FUNCTION_BLOCK EL2596
VAR
	{attribute addProperty Name "WcState"}
	_wcState : WcStateInputToggle;
	{attribute addProperty Name "Info data"}
	_infoData : InfoDataAds;
	_io : EL2596_Data;
END_VAR

PROPERTY IO : REFERENCE TO EL2596_Data
GET
IO REF= _io;
END_GET
END_PROPERTY

PROPERTY WcState : REFERENCE TO WcStateInputToggle
GET
WcState REF= _wcState;
END_GET
END_PROPERTY

END_FUNCTION_BLOCK

(* stored: Version 1.1.0.1, ProductVersion 3.1.4024.9
   POU EL2596: Id {c7ce0382-a06f-0c21-033a-7edddd5a38ea}, SpecialFunc None
   Property IO: Id {ee9ea180-50c2-0d51-3f13-08390b814ded}
   Get Get: Id {2ae2f7f7-b56b-08d0-2934-dd7f30257dd8}
   Property WcState: Id {5fce9226-d75a-0141-3c43-65800f8278cc}
   Get Get: Id {9ab9292c-dbfe-0ecb-277d-4f3cfbca2cfa} *)
